TYPE ZData :
STRUCT
  Config : ZDataConfig;
  Machine : ZDataMachine;
  Calibration : ZDataCalibration;
  Recipe : ZDataRecipe;
END_STRUCT
END_TYPE

(* stored: Version 1.1.0.1
   DUT ZData: Id {02d458ca-eb10-41ad-917a-6c5bc0cc40e5} *)
